// TIA Portal V18 export
// export: Created 2025-12-01T17:50:38.1976771Z, ExportSetting None, DisplayName Totally Integrated Automation Portal, DisplayVersion V18 Update 5, DisplayName TIA Portal Openness, DisplayVersion V18 Update 5, DisplayName TIA Portal Teamcenter Gateway, DisplayVersion V18, DisplayName TIA Portal Version Control Interface, DisplayVersion V18, DisplayName STEP 7 Professional, DisplayVersion V18 Update 5, DisplayName STEP 7 Safety, DisplayVersion V18, DisplayName WinCC Professional, DisplayVersion V18 Update 5
DATA_BLOCK "ST10_Flow12_A2TableUnloading_iDB"   // DB1082
// stored: AutoNumber false, InstanceOfName ST10_Flow12_A2TableUnloading, InstanceOfType FB
"ST10_Flow12_A2TableUnloading"
   // // inherited from GRAPH_BASE
   // VAR_INPUT
   //    iSysInface : "RCS_SysComInterface_V1";
   // END_VAR
   // VAR_IN_OUT
   //    ioPM_Inface : "RCS_PMInterface_V1";
   //    ioStatus : Int;
   // END_VAR
   // VAR
   //    sCtrlMode { S7_SetPoint := 'True'} : "SysFlowCtrlGraph";
   //    sUpdMES_Data : Bool;
   //    工件放行中 : Bool;
   //    前站站号 { ExternalAccessible := 'False'; ExternalVisible := 'False'; ExternalWritable := 'False'} : UInt;
   //    本站站号 { ExternalAccessible := 'False'; ExternalVisible := 'False'; ExternalWritable := 'False'} : UInt;
   //    弹窗Temp : Array[1..10] of Int;
   //    AlarmID : Int;
   //    TON { S7_SetPoint := 'True'} : Array[0..10] of TON_TIME;
   //    TOF { S7_SetPoint := 'True'} : Array[0..10] of TOF_TIME;
   //    sUP { S7_SetPoint := 'True'} : Array[0..10] of Bool;
   //    更新RFID完成 : Bool;
   //    RT_DATA { ExternalAccessible := 'False'; ExternalVisible := 'False'; ExternalWritable := 'False'; S7_SetPoint := 'True'} : G7_RTDataPlus_V6;
   //    Trans1 { ExternalAccessible := 'False'; ExternalVisible := 'False'; ExternalWritable := 'False'; S7_SetPoint := 'True'} : G7_TransitionPlus_V6;
   //    Trans2 { ExternalAccessible := 'False'; ExternalVisible := 'False'; ExternalWritable := 'False'; S7_SetPoint := 'True'} : G7_TransitionPlus_V6;
   //    Trans3 { ExternalAccessible := 'False'; ExternalVisible := 'False'; ExternalWritable := 'False'; S7_SetPoint := 'True'} : G7_TransitionPlus_V6;
   //    Trans325 { ExternalAccessible := 'False'; ExternalVisible := 'False'; ExternalWritable := 'False'; S7_SetPoint := 'True'} : G7_TransitionPlus_V6;
   //    Trans4 { ExternalAccessible := 'False'; ExternalVisible := 'False'; ExternalWritable := 'False'; S7_SetPoint := 'True'} : G7_TransitionPlus_V6;
   //    Trans10 { ExternalAccessible := 'False'; ExternalVisible := 'False'; ExternalWritable := 'False'; S7_SetPoint := 'True'} : G7_TransitionPlus_V6;
   //    Trans102 { ExternalAccessible := 'False'; ExternalVisible := 'False'; ExternalWritable := 'False'; S7_SetPoint := 'True'} : G7_TransitionPlus_V6;
   //    Trans17 { ExternalAccessible := 'False'; ExternalVisible := 'False'; ExternalWritable := 'False'; S7_SetPoint := 'True'} : G7_TransitionPlus_V6;
   //    Trans18 { ExternalAccessible := 'False'; ExternalVisible := 'False'; ExternalWritable := 'False'; S7_SetPoint := 'True'} : G7_TransitionPlus_V6;
   //    Trans19 { ExternalAccessible := 'False'; ExternalVisible := 'False'; ExternalWritable := 'False'; S7_SetPoint := 'True'} : G7_TransitionPlus_V6;
   //    Trans20 { ExternalAccessible := 'False'; ExternalVisible := 'False'; ExternalWritable := 'False'; S7_SetPoint := 'True'} : G7_TransitionPlus_V6;
   //    Trans21 { ExternalAccessible := 'False'; ExternalVisible := 'False'; ExternalWritable := 'False'; S7_SetPoint := 'True'} : G7_TransitionPlus_V6;
   //    Trans22 { ExternalAccessible := 'False'; ExternalVisible := 'False'; ExternalWritable := 'False'; S7_SetPoint := 'True'} : G7_TransitionPlus_V6;
   //    Trans23 { ExternalAccessible := 'False'; ExternalVisible := 'False'; ExternalWritable := 'False'; S7_SetPoint := 'True'} : G7_TransitionPlus_V6;
   //    Trans24 { ExternalAccessible := 'False'; ExternalVisible := 'False'; ExternalWritable := 'False'; S7_SetPoint := 'True'} : G7_TransitionPlus_V6;
   //    Trans30 { ExternalAccessible := 'False'; ExternalVisible := 'False'; ExternalWritable := 'False'; S7_SetPoint := 'True'} : G7_TransitionPlus_V6;
   //    Trans31 { ExternalAccessible := 'False'; ExternalVisible := 'False'; ExternalWritable := 'False'; S7_SetPoint := 'True'} : G7_TransitionPlus_V6;
   //    Trans32 { ExternalAccessible := 'False'; ExternalVisible := 'False'; ExternalWritable := 'False'; S7_SetPoint := 'True'} : G7_TransitionPlus_V6;
   //    Trans200 { ExternalAccessible := 'False'; ExternalVisible := 'False'; ExternalWritable := 'False'; S7_SetPoint := 'True'} : G7_TransitionPlus_V6;
   //    Trans101 { ExternalAccessible := 'False'; ExternalVisible := 'False'; ExternalWritable := 'False'; S7_SetPoint := 'True'} : G7_TransitionPlus_V6;
   //    Trans103 { ExternalAccessible := 'False'; ExternalVisible := 'False'; ExternalWritable := 'False'; S7_SetPoint := 'True'} : G7_TransitionPlus_V6;
   //    Trans106 { ExternalAccessible := 'False'; ExternalVisible := 'False'; ExternalWritable := 'False'; S7_SetPoint := 'True'} : G7_TransitionPlus_V6;
   //    Trans107 { ExternalAccessible := 'False'; ExternalVisible := 'False'; ExternalWritable := 'False'; S7_SetPoint := 'True'} : G7_TransitionPlus_V6;
   //    Trans108 { ExternalAccessible := 'False'; ExternalVisible := 'False'; ExternalWritable := 'False'; S7_SetPoint := 'True'} : G7_TransitionPlus_V6;
   //    Trans109 { ExternalAccessible := 'False'; ExternalVisible := 'False'; ExternalWritable := 'False'; S7_SetPoint := 'True'} : G7_TransitionPlus_V6;
   //    Trans110 { ExternalAccessible := 'False'; ExternalVisible := 'False'; ExternalWritable := 'False'; S7_SetPoint := 'True'} : G7_TransitionPlus_V6;
   //    Trans111 { ExternalAccessible := 'False'; ExternalVisible := 'False'; ExternalWritable := 'False'; S7_SetPoint := 'True'} : G7_TransitionPlus_V6;
   //    Trans283 { ExternalAccessible := 'False'; ExternalVisible := 'False'; ExternalWritable := 'False'; S7_SetPoint := 'True'} : G7_TransitionPlus_V6;
   //    Trans113 { ExternalAccessible := 'False'; ExternalVisible := 'False'; ExternalWritable := 'False'; S7_SetPoint := 'True'} : G7_TransitionPlus_V6;
   //    Trans112 { ExternalAccessible := 'False'; ExternalVisible := 'False'; ExternalWritable := 'False'; S7_SetPoint := 'True'} : G7_TransitionPlus_V6;
   //    Trans115 { ExternalAccessible := 'False'; ExternalVisible := 'False'; ExternalWritable := 'False'; S7_SetPoint := 'True'} : G7_TransitionPlus_V6;
   //    Trans765 { ExternalAccessible := 'False'; ExternalVisible := 'False'; ExternalWritable := 'False'; S7_SetPoint := 'True'} : G7_TransitionPlus_V6;
   //    Trans117 { ExternalAccessible := 'False'; ExternalVisible := 'False'; ExternalWritable := 'False'; S7_SetPoint := 'True'} : G7_TransitionPlus_V6;
   //    Trans766 { ExternalAccessible := 'False'; ExternalVisible := 'False'; ExternalWritable := 'False'; S7_SetPoint := 'True'} : G7_TransitionPlus_V6;
   //    Trans119 { ExternalAccessible := 'False'; ExternalVisible := 'False'; ExternalWritable := 'False'; S7_SetPoint := 'True'} : G7_TransitionPlus_V6;
   //    Trans767 { ExternalAccessible := 'False'; ExternalVisible := 'False'; ExternalWritable := 'False'; S7_SetPoint := 'True'} : G7_TransitionPlus_V6;
   //    Trans768 { ExternalAccessible := 'False'; ExternalVisible := 'False'; ExternalWritable := 'False'; S7_SetPoint := 'True'} : G7_TransitionPlus_V6;
   //    Trans769 { ExternalAccessible := 'False'; ExternalVisible := 'False'; ExternalWritable := 'False'; S7_SetPoint := 'True'} : G7_TransitionPlus_V6;
   //    Trans770 { ExternalAccessible := 'False'; ExternalVisible := 'False'; ExternalWritable := 'False'; S7_SetPoint := 'True'} : G7_TransitionPlus_V6;
   //    Trans124 { ExternalAccessible := 'False'; ExternalVisible := 'False'; ExternalWritable := 'False'; S7_SetPoint := 'True'} : G7_TransitionPlus_V6;
   //    Trans125 { ExternalAccessible := 'False'; ExternalVisible := 'False'; ExternalWritable := 'False'; S7_SetPoint := 'True'} : G7_TransitionPlus_V6;
   //    Trans771 { ExternalAccessible := 'False'; ExternalVisible := 'False'; ExternalWritable := 'False'; S7_SetPoint := 'True'} : G7_TransitionPlus_V6;
   //    Trans127 { ExternalAccessible := 'False'; ExternalVisible := 'False'; ExternalWritable := 'False'; S7_SetPoint := 'True'} : G7_TransitionPlus_V6;
   //    Trans128 { ExternalAccessible := 'False'; ExternalVisible := 'False'; ExternalWritable := 'False'; S7_SetPoint := 'True'} : G7_TransitionPlus_V6;
   //    Trans129 { ExternalAccessible := 'False'; ExternalVisible := 'False'; ExternalWritable := 'False'; S7_SetPoint := 'True'} : G7_TransitionPlus_V6;
   //    Trans130 { ExternalAccessible := 'False'; ExternalVisible := 'False'; ExternalWritable := 'False'; S7_SetPoint := 'True'} : G7_TransitionPlus_V6;
   //    Trans131 { ExternalAccessible := 'False'; ExternalVisible := 'False'; ExternalWritable := 'False'; S7_SetPoint := 'True'} : G7_TransitionPlus_V6;
   //    Trans132 { ExternalAccessible := 'False'; ExternalVisible := 'False'; ExternalWritable := 'False'; S7_SetPoint := 'True'} : G7_TransitionPlus_V6;
   //    Trans133 { ExternalAccessible := 'False'; ExternalVisible := 'False'; ExternalWritable := 'False'; S7_SetPoint := 'True'} : G7_TransitionPlus_V6;
   //    Trans134 { ExternalAccessible := 'False'; ExternalVisible := 'False'; ExternalWritable := 'False'; S7_SetPoint := 'True'} : G7_TransitionPlus_V6;
   //    Trans135 { ExternalAccessible := 'False'; ExternalVisible := 'False'; ExternalWritable := 'False'; S7_SetPoint := 'True'} : G7_TransitionPlus_V6;
   //    Trans139 { ExternalAccessible := 'False'; ExternalVisible := 'False'; ExternalWritable := 'False'; S7_SetPoint := 'True'} : G7_TransitionPlus_V6;
   //    Trans140 { ExternalAccessible := 'False'; ExternalVisible := 'False'; ExternalWritable := 'False'; S7_SetPoint := 'True'} : G7_TransitionPlus_V6;
   //    Trans146 { ExternalAccessible := 'False'; ExternalVisible := 'False'; ExternalWritable := 'False'; S7_SetPoint := 'True'} : G7_TransitionPlus_V6;
   //    Trans250 { ExternalAccessible := 'False'; ExternalVisible := 'False'; ExternalWritable := 'False'; S7_SetPoint := 'True'} : G7_TransitionPlus_V6;
   //    Trans613 { ExternalAccessible := 'False'; ExternalVisible := 'False'; ExternalWritable := 'False'; S7_SetPoint := 'True'} : G7_TransitionPlus_V6;
   //    F12_Initial { ExternalAccessible := 'False'; ExternalVisible := 'False'; ExternalWritable := 'False'; S7_SetPoint := 'True'} : G7_StepPlus_V6;
   //    S2 { ExternalAccessible := 'False'; ExternalVisible := 'False'; ExternalWritable := 'False'; S7_SetPoint := 'True'} : G7_StepPlus_V6;
   //    S3 { ExternalAccessible := 'False'; ExternalVisible := 'False'; ExternalWritable := 'False'; S7_SetPoint := 'True'} : G7_StepPlus_V6;
   //    S4 { ExternalAccessible := 'False'; ExternalVisible := 'False'; ExternalWritable := 'False'; S7_SetPoint := 'True'} : G7_StepPlus_V6;
   //    S5_MESInitial { ExternalAccessible := 'False'; ExternalVisible := 'False'; ExternalWritable := 'False'; S7_SetPoint := 'True'} : G7_StepPlus_V6;
   //    "ServoReady?" { ExternalAccessible := 'False'; ExternalVisible := 'False'; ExternalWritable := 'False'; S7_SetPoint := 'True'} : G7_StepPlus_V6;
   //    WaitRobotInitialFinish { ExternalAccessible := 'False'; ExternalVisible := 'False'; ExternalWritable := 'False'; S7_SetPoint := 'True'} : G7_StepPlus_V6;
   //    S10_InitialFinish { ExternalAccessible := 'False'; ExternalVisible := 'False'; ExternalWritable := 'False'; S7_SetPoint := 'True'} : G7_StepPlus_V6;
   //    "Servo returns to1st Pos" { ExternalAccessible := 'False'; ExternalVisible := 'False'; ExternalWritable := 'False'; S7_SetPoint := 'True'} : G7_StepPlus_V6;
   //    ServoPosCount { ExternalAccessible := 'False'; ExternalVisible := 'False'; ExternalWritable := 'False'; S7_SetPoint := 'True'} : G7_StepPlus_V6;
   //    ServoPosCountJudge { ExternalAccessible := 'False'; ExternalVisible := 'False'; ExternalWritable := 'False'; S7_SetPoint := 'True'} : G7_StepPlus_V6;
   //    ServoPosCountClear { ExternalAccessible := 'False'; ExternalVisible := 'False'; ExternalWritable := 'False'; S7_SetPoint := 'True'} : G7_StepPlus_V6;
   //    CountCompare { ExternalAccessible := 'False'; ExternalVisible := 'False'; ExternalWritable := 'False'; S7_SetPoint := 'True'} : G7_StepPlus_V6;
   //    TableLackMaterial { ExternalAccessible := 'False'; ExternalVisible := 'False'; ExternalWritable := 'False'; S7_SetPoint := 'True'} : G7_StepPlus_V6;
   //    WaitFixtureScanFinish { ExternalAccessible := 'False'; ExternalVisible := 'False'; ExternalWritable := 'False'; S7_SetPoint := 'True'} : G7_StepPlus_V6;
   //    ResetPartMissingAlarm { ExternalAccessible := 'False'; ExternalVisible := 'False'; ExternalWritable := 'False'; S7_SetPoint := 'True'} : G7_StepPlus_V6;
   //    ProcessStart { ExternalAccessible := 'False'; ExternalVisible := 'False'; ExternalWritable := 'False'; S7_SetPoint := 'True'} : G7_StepPlus_V6;
   //    WaitChangeOverFinish { ExternalAccessible := 'False'; ExternalVisible := 'False'; ExternalWritable := 'False'; S7_SetPoint := 'True'} : G7_StepPlus_V6;
   //    WaitServoInPosition { ExternalAccessible := 'False'; ExternalVisible := 'False'; ExternalWritable := 'False'; S7_SetPoint := 'True'} : G7_StepPlus_V6;
   //    "Detect cartridge exist" { ExternalAccessible := 'False'; ExternalVisible := 'False'; ExternalWritable := 'False'; S7_SetPoint := 'True'} : G7_StepPlus_V6;
   //    "Detect Ring exist" { ExternalAccessible := 'False'; ExternalVisible := 'False'; ExternalWritable := 'False'; S7_SetPoint := 'True'} : G7_StepPlus_V6;
   //    "Detect UnloadingRing exist" { ExternalAccessible := 'False'; ExternalVisible := 'False'; ExternalWritable := 'False'; S7_SetPoint := 'True'} : G7_StepPlus_V6;
   //    "Detect UnloadingRing exist_1" { ExternalAccessible := 'False'; ExternalVisible := 'False'; ExternalWritable := 'False'; S7_SetPoint := 'True'} : G7_StepPlus_V6;
   //    PartMissingAlarm { ExternalAccessible := 'False'; ExternalVisible := 'False'; ExternalWritable := 'False'; S7_SetPoint := 'True'} : G7_StepPlus_V6;
   //    Step111 { ExternalAccessible := 'False'; ExternalVisible := 'False'; ExternalWritable := 'False'; S7_SetPoint := 'True'} : G7_StepPlus_V6;
   //    "Request robot pick" { ExternalAccessible := 'False'; ExternalVisible := 'False'; ExternalWritable := 'False'; S7_SetPoint := 'True'} : G7_StepPlus_V6;
   //    SensorNoPart { ExternalAccessible := 'False'; ExternalVisible := 'False'; ExternalWritable := 'False'; S7_SetPoint := 'True'} : G7_StepPlus_V6;
   //    CountClear { ExternalAccessible := 'False'; ExternalVisible := 'False'; ExternalWritable := 'False'; S7_SetPoint := 'True'} : G7_StepPlus_V6;
   //    CountClear_1 { ExternalAccessible := 'False'; ExternalVisible := 'False'; ExternalWritable := 'False'; S7_SetPoint := 'True'} : G7_StepPlus_V6;
   //    "A-Loading-02UpDownTakeCylinderToWP" { ExternalAccessible := 'False'; ExternalVisible := 'False'; ExternalWritable := 'False'; S7_SetPoint := 'True'} : G7_StepPlus_V6;
   //    "CheckA-Loading-02HorizontalCylinderPos" { ExternalAccessible := 'False'; ExternalVisible := 'False'; ExternalWritable := 'False'; S7_SetPoint := 'True'} : G7_StepPlus_V6;
   //    "A-Loading-02UpDownTakeCylinderToWP_1" { ExternalAccessible := 'False'; ExternalVisible := 'False'; ExternalWritable := 'False'; S7_SetPoint := 'True'} : G7_StepPlus_V6;
   //    "A-Loading-02HorizontalCylinderToHP" { ExternalAccessible := 'False'; ExternalVisible := 'False'; ExternalWritable := 'False'; S7_SetPoint := 'True'} : G7_StepPlus_V6;
   //    "A-Loading-02UpDownTakeCylinderToHP_2" { ExternalAccessible := 'False'; ExternalVisible := 'False'; ExternalWritable := 'False'; S7_SetPoint := 'True'} : G7_StepPlus_V6;
   //    "A-Loading-02HorizontalCylinderToWP_1" { ExternalAccessible := 'False'; ExternalVisible := 'False'; ExternalWritable := 'False'; S7_SetPoint := 'True'} : G7_StepPlus_V6;
   //    "A-Loading-02UpDownTakeCylinderToHP3" { ExternalAccessible := 'False'; ExternalVisible := 'False'; ExternalWritable := 'False'; S7_SetPoint := 'True'} : G7_StepPlus_V6;
   //    TimDelay { ExternalAccessible := 'False'; ExternalVisible := 'False'; ExternalWritable := 'False'; S7_SetPoint := 'True'} : G7_StepPlus_V6;
   //    TimDelay_1 { ExternalAccessible := 'False'; ExternalVisible := 'False'; ExternalWritable := 'False'; S7_SetPoint := 'True'} : G7_StepPlus_V6;
   //    "A-Loading-02HorizontalCylinderToHP_1" { ExternalAccessible := 'False'; ExternalVisible := 'False'; ExternalWritable := 'False'; S7_SetPoint := 'True'} : G7_StepPlus_V6;
   //    ServoNeedMove { ExternalAccessible := 'False'; ExternalVisible := 'False'; ExternalWritable := 'False'; S7_SetPoint := 'True'} : G7_StepPlus_V6;
   //    "No cartridge" { ExternalAccessible := 'False'; ExternalVisible := 'False'; ExternalWritable := 'False'; S7_SetPoint := 'True'} : G7_StepPlus_V6;
   //    "No Ring" { ExternalAccessible := 'False'; ExternalVisible := 'False'; ExternalWritable := 'False'; S7_SetPoint := 'True'} : G7_StepPlus_V6;
   //    "Clearing mode?" { ExternalAccessible := 'False'; ExternalVisible := 'False'; ExternalWritable := 'False'; S7_SetPoint := 'True'} : G7_StepPlus_V6;
   //    "Wait  robot finish task" { ExternalAccessible := 'False'; ExternalVisible := 'False'; ExternalWritable := 'False'; S7_SetPoint := 'True'} : G7_StepPlus_V6;
   //    WaitChangeOverOK { ExternalAccessible := 'False'; ExternalVisible := 'False'; ExternalWritable := 'False'; S7_SetPoint := 'True'} : G7_StepPlus_V6;
   //    WaitEmptyFinish { ExternalAccessible := 'False'; ExternalVisible := 'False'; ExternalWritable := 'False'; S7_SetPoint := 'True'} : G7_StepPlus_V6;
   //    "Process Finish" { ExternalAccessible := 'False'; ExternalVisible := 'False'; ExternalWritable := 'False'; S7_SetPoint := 'True'} : G7_StepPlus_V6;
   // END_VAR
BEGIN
END_DATA_BLOCK
